Yaskawa INFORM job: JOBDONE.JBI

/JOB
//NAME JOBDONE
//POS
///NPOS 0,0,0,0,0,0
//INST
///DATE 2018/11/28 10:49
///ATTR SC,RW,MC
NOP
DOUT OT#(578) OFF
TIMER T=0.50
WAIT IG#(76)=0
WAIT IG#(75)=0
DOUT OT#(579) ON
WAIT IN#(579)=ON
DOUT OT#(579) OFF
END
